PROGRAM MAIN
VAR
	increment 	AT %I*	: INT 	:= 0;
	sum 		AT %Q*	: INT	:= 0;
END_VAR

sum := sum + increment;

END_PROGRAM

(* stored: Version 1.1.0.1, ProductVersion 3.1.4024.10
   POU MAIN: Id {05518f30-63f5-43e5-a500-2e4c842868d1}, SpecialFunc None *)
